{attribute 'GeneratedUsingTerminal: EL4022-0000-0018'}
{attribute addProperty BoxType "EL4022-0000-0018"}
{attribute addProperty Description "EL4022 2Ch. Ana. Output 4-20mA, 12bit"}
{attribute addProperty Physics "KK"}
{attribute addProperty Id "AO_Output_Channel_1AT %Q*AO_Output_Channel_BA7EBB7C2AO_Output_Channel_2AT %Q*AO_Output_Channel_BA7EBB7C2WcStateAT %I*WcState_0B2B16F91InfoDataAT %I*InfoData_32EB74EA10"}
{attribute addProperty CRC "1524858257"}
{attribute addProperty Size "15"}
TYPE EL4022_5AE37D91 EXTENDS EtcSlaveTerminalBase_947E5A46 :
STRUCT
	{attribute addProperty Name "AO_Output_Channel_1"}
	AO_Output_Channel_1 : AO_Output_Channel_BA7EBB7C;
	{attribute addProperty Name "AO_Output_Channel_2"}
	AO_Output_Channel_2 : AO_Output_Channel_BA7EBB7C;
	{attribute addProperty Name "WcState"}
	WcState : WcState_0B2B16F9;
	{attribute addProperty Name "InfoData"}
	InfoData : InfoData_32EB74EA;
END_STRUCT
END_TYPE

(* stored: Version 1.2.0.0, ProductVersion 3.1.4024.9
   DUT EL4022_5AE37D91: Id {7a32dc13-e5a6-4ccb-8152-3710e0be90dc} *)
